(*
Nazwa:			FB_ROPPCapping
Opis:			
Wersja:			v0.1
Data:			2025-01-13
Autor:			DP
Urzadzenia:		
Konfiguracja:	
Info:
-
*)

FUNCTION_BLOCK FB_ROPPCapping
VAR_INPUT
	
	bEnable						: BOOL;					//Zezowlenie na pracę stacji sprawdzania
	bEStop						: BOOL;					//Stop Awaryjny nieaktywny
	bRun1						: BOOL;					//Włączenie 
	bRun2						: BOOL;					//Włączenie
	bRunEngine					: BOOL;					
	bHoming						: BOOL;					//Zezwolenie na wykonanie bazowania i pozycjonowania stacji sprawdzania
	bHeightSet					: BOOL;					//Bit do bazowania stacji na ustaloną wysokość 
	bIgnoreError				: BOOL;					//Ignorowania błędów cyklu pracy
	bReset						: BOOL;					//Reset błędu, jeśli w stanie "eError"
	iTime						: INT; 				
	iTime2						: INT; 				
	iTool						: INT;					//Wybór narzędzia (1-5), opisy w tablicy AsGripperScrewerTool	

	IbCapping1Tool1ActuatorUpSensor		: BOOL;		
	IbCapping1Tool1ActuatorDownSensor	: BOOL;	
	IbCapping2Tool1ActuatorUpSensor		: BOOL;	
	IbCapping2Tool1ActuatorDownSensor	: BOOL;	

	IbCapping1Tool2ActuatorUpSensor		: BOOL;		
	IbCapping1Tool2ActuatorCappingDoneSensor: BOOL;	
	IbCapping2Tool2ActuatorUpSensor			: BOOL;	
	IbCapping2Tool2ActuatorCappingDoneSensor: BOOL;	



	InEngineVelocityCV 			: UDINT;		
	InEngineSTW 				: UINT; 				// Statusword transportera wejściowo wyjściowego
	IbEngineWcState				: BOOL; 				// Statusword transportera wejściowo wyjściowego
	InEngine2VelocityCV 		: UDINT;		
	InEngine2STW 				: UINT; 				// Statusword transportera wejściowo wyjściowego
	IbEngine2WcState			: BOOL; 				// Statusword transportera wejściowo wyjściowego

	_HEIGHTMOTOR_ 				: BOOL;
	lrHeightMotorSV				: LREAL;			// Zadana wysokość
	udiHeightMotorEncoderCV		: UDINT;				// Ilość impulsów z modułu enkoderowego
	bHeightEncoderSetCDone		: BOOL;					// Zerowanie enkodera wykonane
	rHeightMotorPositionOffset 	: REAL;					// Wysokość bazowani podnośnika
	lrMaxHeight					: LREAL;				// Maksymalna wysokość podnośnika 
	lrMinHeight					: LREAL;				// Minimalna wysokość podnośnika

	bManualMovement				: BOOL; 				//Uruchomienie trybu ruchów ręcznych
	udiStationIndex				: UDINT;				// Indywidualny numer stacji
	sStationName				: STRING;				// Nazwa stacji
	
END_VAR

VAR_OUTPUT
	eState						: E_Station;			// Aktualny stan stacju
	eRunningState				: E_GripperScrewer;		// Stan pracy stacji
	eRunningStateBeforeEstop	: E_GripperScrewer;  	// Stan przed Estope
	bError						: BOOL;					// Błąd stacji
	udiErrorID					: UDINT;				// Nr blędu przeciągania formatek
	sErrorDescription			: STRING(200);			// Opis błędu
	sErrorDescription2			: STRING(200);			// Opis błędu
	sErrorStationName			: STRING;				// Nazwa stacj
	udiStationID				: UDINT;				// Nr stacji

	bHeightMotorUp				: BOOL;					//Sterowanie silnikiem podnośnika  - RUCH W GÓRĘ
	bHeightMotorDown			: BOOL;					//Sterowanie silnikiem podnośnika  - RUCH W DÓŁ
	udiHeightMotorEncoderSetCV	: UDINT;		
	bHeightEncoderSetC			: BOOL;					// Zerowanie enkodera
	lrHeightMotorCV				: LREAL;				// Aktualna pozycja podnośnika

	QnEngineVelocitySV 			: UDINT; 				// Nastawa prędkości
	QnEngineCTW 				: UINT;  				// Controlword transportera we/wy	
	QnEngine2VelocitySV 		: UDINT; 				// Nastawa prędkości
	QnEngine2CTW 				: UINT;  				// Controlword transportera we/wy	
	bHomingNeeded				: BOOL;					// Wymagane ponowne bazowanie (blad podczas bazowania lub stop awaryjny)
	bHomingDone					: BOOL;					// Stacja zbazowana 
	bCycleDone1					: BOOL;					// Sygnał o zakończeniu cyklu
	bCycleNotDone1				: BOOL;					// Sygnał o niezakończonym cyklu	
	bCycleDone2					: BOOL;					// Sygnał o zakończeniu cyklu
	bCycleNotDone2				: BOOL;					// Sygnał o niezakończonym cyklu

	tCycleTime					: TIME;	 				// Czas cyklu 
	sWarningDescription			: STRING;
	bWarning1					: BOOL;
	udiWarningID				: UDINT;
	
	bCapping1Tool1Actuator		: BOOL;
	bCapping2Tool1Actuator		: BOOL;
	bCapping12Tool1BlockActuator: BOOL;
	bCappingBlockActuator		: BOOL;
	bCapping1Tool2Down			: BOOL;		
	bCapping1Tool2Tight			: BOOL;	
	bCapping1Tool2Realese		: BOOL;	
	bCapping2Tool2Down			: BOOL;		
	bCapping2Tool2Tight			: BOOL;	
	bCapping2Tool2Realese		: BOOL;
	bFormPositioning			: BOOL;

	AsToolDescription			: ARRAY [1..10] OF STRING;	// Opis narzędzi, 1 - Opis narzędzia nr 1, 2 - Opis narzędzia nr 2
	sTool						: STRING;
	
END_VAR

VAR_IN_OUT
	
	bManualHeightMotorUp				: BOOL;					//Ruch ręczny podnośnika stacji w górę
	bManualHeightMotorDown				: BOOL;					//Ruch ręczny podnośnika stacji w dół
	bManualEngine1						: BOOL;					//Ręczne włączenie silnika sortera
	bManualEngine2						: BOOL;					//Ręczne włączenie silnika sortera
	bManualCapping1Tool1Actuator		: BOOL;
	bManualCapping2Tool1Actuator		: BOOL;
	bManualCapping12Tool1BlockActuator	: BOOL;
	bManualCappingBlockActuator			: BOOL;
	bManualCapping1Tool2Down			: BOOL;		
	bManualCapping1Tool2Tight			: BOOL;	
	bManualCapping1Tool2Realese			: BOOL;	
	bManualCapping2Tool2Down			: BOOL;		
	bManualCapping2Tool2Tight			: BOOL;	
	bManualCapping2Tool2Realese			: BOOL;
	bManualFormPositioning				: BOOL;

END_VAR

VAR
	i							:	INT;
	aBufferedSensorValue		:	ARRAY[0..50] OF BOOL;	
	iValvesCycleCase			:	INT;
	rtOutSensor					:	R_TRIG;

	// State
	eLastState					: E_Station;			//Stan ogólny bloku
	eLastStateTemp				: E_Station;			//Stan ogólny bloku
	eLastRunningState			: E_GripperScrewer;		//Stan podbloku
	eLastRunningStateTemp		: E_GripperScrewer;		//Stan podbloku

	fbHeightMotorEncoder		: FB_JiesangActuatorEncoderModul;				// Blok enkodera podnośnika chwytaka stabilizującego pod zakręcarką	
	bHeightMotorEncoderCounterReset						:BOOL; 				// Sygnał resetu enkodera
	lrLastHeightMotorPositionCV		: LREAL;				// Pozycja podnośnika w poprzednim cyklu programu
	bHeightMotorEncoderHomed	: BOOL;					// Informacja od enkodera że jest zbazowany		
	bStateError					: BOOL;
	
	tofHeightMotorDown			: TOF;					// Opóźnienie ruchu w dół, żeby nie przeciązać rozruchem układu
	rtEncoderHomed				: R_TRIG;				// Bit zakończenia enkodera
		
	tonHeightNoChange			: TON; 					// Timer wykrycia braku ruchu siłownika zmiany wysokości stacji
	tonHeightNoChangeTime		: TON; 					// Timer wykrycia braku ruchu siłownika zmiany wysokości stacji
	
	tonLimitPosMinReachedDelay	: TON;					// Timer osoiągniecia minimalnej wyskości 
	tonLimitPosMaxReachedDelay	: TON;					// Timer osiągnięcia maksymalnej wyskości
	tonSortingEngineOn			: TON;					// Opóźnienie po załączeniu napędu
	tonSortingEngineOff			: TON;					// Opóźnienie wyłączenia napędu
	tonSleeveFullEngineOn		: TON;					// Czas załączenia napędu po wykrciu braku nasadek
	tonEngineBlocked			: TON;					// Zablokowany silnik	
	rtCapSorterSensor			: R_TRIG;				// Triger
	tonTryUnblockWheel			: TON;					// Czas ruchu falownika w drugą stronę
	tofCapFeederSorterCapSensor	: TOF;					// Opóźnienie sygnału z czujnika obecności nasadki ultradzwiek
	tonCapFeederSorterCapSensor	: TON;					// Opóźnienie sygnału z czujnika obecności nasadki ultradźwięk
	tonAirBeforeStart			: TON;					// Czasówka opóźeniani przedmuchu
	tonAirBeforeStart2			: TON;					// Czasówka opóźeniani przedmuchu
	tonAirAfterStop				: TON;					// Czasówka przedmuchu po zatrzymaniu
	tonStoppingTime				: TON;					// Czasówka zbyt długiego zatrzymawania

	
	tonErrorHeightChange		: TON; 					// Timer błędu zacięcia się podnośnika
	tonMaxHeightError			: TON;					// Timer ustawienia zbyt dużej wysokości stacji
	tonMinHeightError			: TON;					// Timer ustawienia zbyt małej wysokości stacji
	tonCycleTimer				: TON;					// Czasówka cyklu
	rtrigCycleTimerRead			: R_TRIG;				// Trigger do statystyk cyklu 
	
	rtResetCommands				: R_TRIG;
	tonHomingSensor: TON;
	TimerOn: TON;
	TimerOff: TON;
	bImpOn: BOOL;
	rtCapFeederSorterCapSensor: R_TRIG;
	bBlowDelay: BOOL;
	tonbBlowDelay: TON;
	
	fbInverter: FB_MitsubishiInverter;
	fbInverter2: FB_MitsubishiInverter;	
	tonInverterError: TON;
	tonInverter2Error: TON;	
	tonbCapping1Tool2ActuatorUpError: TON;
	tonbCapping2Tool2ActuatorUpError: TON;	
	
	(*Ostrzeżenia*)
	fbbLevelSensor:	FB_InputFilter;
	(*Inne*)	

	tonGates1	:	TON;	//Czasówka dla szlabanów w rękawe
	tonGates2	:	TON;	//Czasówka dla szlabanów w rękawe
	tonGates3	:	TON;	//Czasówka dla szlabanów w rękawe
	tonGates4	:	TON;	//Czasówka dla szlabanów w rękawe

	toneHolding1 :TON;
	toneHolding2 :TON;
	toneGoingUp	:TON;
	toneHolding1Tool2 :TON;
	toneHolding2Tool2 :TON;
	
	bDone1				: BOOL;					// Sygnał o niezakończonym cyklu
	bDone2				: BOOL;					// Sygnał o niezakończonym cyklu
	
	tonDown1:TON;
	tonDown2:TON;	
	tonEnginesRun:TON;	
	tonDone	:TON;	
	ftbRunEngine: F_TRIG;
	bGates	    :	BOOL;	//Controla szłabanow w rękawe  
	bTryUnblockWheel : BOOL;
	iTryUnblockWheel : INT;
END_VAR

//Wywołanie bloczków od stacji. Ważna jest ich kolejność!!!
ACT_Limits();
ACT_HeightMotor();
ACT_ErrorHandling();

ACT_Signals();
ACT_Control();
aEngine();
ACT_Inverter();
ACT_Statistic();
ACT_Status();
ACT_Warnings();
aStationID();	

lrLastHeightMotorPositionCV:=lrHeightMotorCV;

ACTION ACT_Control:
	(*****Wyłączenie enable*****)
	IF NOT bEnable THEN
		IF eState <> E_Station.eDisabled AND eState <> E_Station.ePreparingToDisable THEN
				eState 				:= E_Station.ePreparingToDisable; 
		END_IF	
	END_IF

	(*****Estop*****)
	IF NOT bEstop  THEN	
		IF eState <> E_Station.eAborted AND eState <> E_Station.eAborting AND eState <> E_Station.eDisabled THEN
				eState 				:= E_Station.eAborting; 
		END_IF
	END_IF


	CASE eState OF
//--------------------------------------------------------------------------------
// Stan maszyny po wyłączeniu i przygotowanie do uruchomienia
	E_Station.eDisabled: 					// Stan nieaktywnosci (Stacja wyłączona) 
	
		IF bEnable THEN
			eState 				:= E_Station.ePreparingToReady; 
		END_IF 
		
//--------------------------------------------------------------------------------
// Stan maszyny po zatrzymaniu awaryjnym   
	E_Station.eAborted: 					// Stan bezpiecznego zatrzymania (po Abortingu) 

		IF bEStop THEN
			eState 				:= E_Station.ePreparingToReady;
		END_IF
		
//--------------------------------------------------------------------------------
// Stan maszyny naciśnieciu estopa 	
	E_Station.eAborting:                 	// Stan bezpiecznego zatrzymywania (po EStopie)

		ACT_ResetCommands();

		eState 						:=  E_Station.eAborted;  
		eRunningState				:=	E_GripperScrewer.eReady;
		
//--------------------------------------------------------------------------------
// Stan masyzny po wykryciu błędu			
	E_Station.eError:                 	 	// Stan błędu 	
		
		ACT_ResetCommands();
		
		IF bReset THEN
			eState 					:= E_Station.eResetting;
			bError					 := FALSE;
		END_IF
		
//--------------------------------------------------------------------------------
// Stan masyzny po wykryciu błędu
	E_Station.eResetting:					// Stan resetowania bledu (po Errorze)
			CASE udiErrorID OF
		
				//Error - Błąd falownika
				353,354:
					fbInverter.bReset	:= TRUE;
					fbInverter2.bReset	:= TRUE;					
					bError 				:= FALSE;
				ELSE
					bError := FALSE;	
			END_CASE		
		
		IF NOT bError AND fbInverter.eState = E_Station.eReady THEN
			fbInverter.bReset	:= FALSE;	
			fbInverter2.bReset	:= FALSE;
			//{warning 'Sprawdzić błąd falownika CapFeeder'}
			udiErrorID 			:=	0;
			sErrorDescription 	:=	'';
			eState 				:=	E_Station.ePreparingToReady;
			eRunningState		:=	E_GripperScrewer.eReady;
		ELSE
			eState 				:=	E_Station.eError;
		END_IF
    
//--------------------------------------------------------------------------------
// Stan ruchoow manualnych
	E_Station.eManualMovement:     			// Stan ruchów manualnych  
   
		ACT_ManualMovements();
		//Wyjście z trybu serwisowego
		IF NOT bManualMovement THEN
			bHeightMotorUp				:=	FALSE;
			bHeightMotorDown			:=	FALSE;
			eState:=E_Station.eReady;
		END_IF
		
//--------------------------------------------------------------------------------
// Stan rozpoczecia bazowania
	E_Station.eHoming:						// Stan bazowania 
		
		ACT_Homing();
		IF NOT bHoming AND NOT bHeightSet THEN
			bHeightMotorDown				:=	FALSE;
			bHeightMotorUp					:=	FALSE;
		   eState							:=	E_Station.ePreparingToReady;
		END_IF		
		
//--------------------------------------------------------------------------------
// Stan zakończenia bazowania
	E_Station.eHomingDone:                  // Stan wykonania bazowania 
	
		bHeightMotorDown					:=	FALSE;
		bHeightMotorUp						:=	FALSE;
		bHeightMotorEncoderCounterReset		:=	FALSE;
		bHomingDone							:=	TRUE;
		IF NOT bHoming AND NOT bHeightSet THEN
		   eState:=E_Station.eReady;
		END_IF
		
//--------------------------------------------------------------------------------
// Stan przygotowania do gotowości
	E_Station.ePreparingToReady:            // Stan przygotowywania do gotowosci (zawsze przed Ready)  

		eRunningState	:=	E_GripperScrewer.eReady;
		eState			:=	E_Station.eReady;	
		
//-------------------------------------------------------------------------------
// Stan przygotowania do wyłączenia maszyny
	E_Station.ePreparingToDisable:          // Stan przygotowywania do nieaktywnosci (po wyłączeniu Enable) 

		bHeightMotorUp		:=	TRUE;
		bHeightMotorDown	:=	FALSE;	
		IF tonHeightNoChange.Q OR tonHeightNoChangeTime.Q THEN
			bHeightMotorUp			:=	FALSE;
			bHeightMotorDown		:=	FALSE;	
			eRunningState			:=	E_GripperScrewer.eReady;		
			eState					:=	E_Station.eDisabled;
		END_IF	
			
//--------------------------------------------------------------------------------
// Stan gotowości
	E_Station.eReady:						// Stan gotowosci 
	
		(*Skasowanie wszystkich komend*)
		IF rtResetCommands.Q THEN	ACT_ResetCommands();	END_IF
	
		IF (bRun1 OR bRun2) AND NOT bCycleDone1 AND NOT bCycleNotDone1 AND NOT bCycleDone2 AND NOT bCycleNotDone2 THEN
			eState 				:= E_Station.eStarting; 
		END_IF
		IF bHoming OR bHeightSet THEN
			eState 				:= E_Station.eHoming; 
		END_IF
		IF bManualMovement THEN
			bManualHeightMotorUp					:=	bHeightMotorUp;					
			bManualHeightMotorDown				:=	bHeightMotorDown;	
			bManualEngine1						:=	fbInverter.bRun;							
			bManualEngine2						:=	fbInverter2.bRun;		
			bManualCapping1Tool1Actuator		:=	bCapping1Tool1Actuator;		
			bManualCapping2Tool1Actuator		:=	bCapping2Tool1Actuator;		
			bManualCapping12Tool1BlockActuator	:=	bCapping12Tool1BlockActuator;
			bManualCappingBlockActuator			:=	bCappingBlockActuator;	
			bManualCapping1Tool2Down			:=	bCapping1Tool2Down;	
			bManualCapping1Tool2Tight			:=	bCapping1Tool2Tight;			
			bManualCapping1Tool2Realese			:=	bCapping1Tool2Realese;		
			bManualCapping2Tool2Down			:=	bCapping2Tool2Down;				
			bManualCapping2Tool2Tight			:=	bCapping2Tool2Tight;
			bManualCapping2Tool2Realese			:=	bCapping2Tool2Realese;
			bManualFormPositioning				:=	bFormPositioning;			
			eState 								:=	E_Station.eManualMovement; 
		END_IF
		IF NOT bRun1 AND NOT bRun2 THEN
			bDone1						:= FALSE;
			bDone2						:= FALSE;
			bCycleDone1 				:= FALSE;
			bCycleNotDone1 				:= FALSE;	
			bCycleDone2					:= FALSE;
			bCycleNotDone2 				:= FALSE;	
			bWarning1					:= FALSE;	
		END_IF
		
//--------------------------------------------------------------------------------
// Stan zatrzymywania
	E_Station.eStopping:					// Stan zatrzymywania 
		
		ACT_Running();

		IF tonStoppingTime.Q THEN
			ACT_ResetCommands();
			eRunningState							:= E_GripperScrewer.eReady;
			eState									:= E_Station.eReady;
		END_IF

		
//--------------------------------------------------------------------------------
// Stan uruchomienia lini ( po eReady)
	E_Station.eStarting:                  	// Stan uruchamiania (po Ready)

		eState					 := E_Station.eRunning; 

//--------------------------------------------------------------------------------
// Stan wykonywania pracy
	E_Station.eRunning:               		// Stan wykonywania cyklu (po Startingu), w tym stanie osobny

		ACT_Running();
		IF NOT bRun1 AND NOT bRun2 THEN					(*Przerywanie cyklu*)
			eState 				 := E_Station.eStopping;	
		END_IF
		IF (bCycleDone1 OR bCycleNotDone1) AND (bCycleDone2 OR bCycleNotDone2)  THEN (*Cykl zakończony*)
			eState 				 := E_Station.eReady;
		END_IF						
		
		
END_CASE
END_ACTION

ACTION ACT_ErrorHandling:
//OBSŁUGA BŁĘDÓW STACJI SPRAWDZANIA
//************LISTA BŁĘDÓW***************
bStateError:= (eState=E_Station.eError) OR (eState=E_Station.eResetting) OR bIgnoreError;
//************LISTA BŁĘDÓW***************

//Error 1 - podnośnik nie porusza się pomimo wysterowania 
tonErrorHeightChange(IN:=(bHeightMotorUp OR bHeightMotorDown) AND lrLastHeightMotorPositionCV=lrHeightMotorCV, PT:=T#3S);
tonMaxHeightError	(IN:=lrHeightMotorSV>lrMaxHeight AND NOT bHomingNeeded AND eState=E_Station.eReady,PT:=T#30S);
tonMinHeightError	(IN:=lrHeightMotorSV<lrMinHeight AND NOT bHomingNeeded AND eState=E_Station.eReady,PT:=T#30S);
tonInverterError	(IN:=fbInverter.bError AND NOT bStateError, PT:=T#3S);
tonInverter2Error	(IN:=fbInverter2.bError AND NOT bStateError, PT:=T#3S);

tonbCapping1Tool2ActuatorUpError (IN:= iTool = 2 (*G.dociskająca*) AND NOT IbCapping1Tool2ActuatorUpSensor AND NOT bCapping1Tool2Down, PT:=T#2S);
tonbCapping2Tool2ActuatorUpError (IN:= iTool = 2 (*G.dociskająca*) AND NOT IbCapping2Tool2ActuatorUpSensor AND NOT bCapping2Tool2Down, PT:=T#2S);

IF (bEnable OR (eState = E_Station.ePreparingToDisable)) AND NOT bIgnoreError THEN
	
	IF tonErrorHeightChange.Q THEN
		bError:=TRUE;
		udiErrorID:=350;
		sErrorDescription:='Blokada podnośnika lub brak zasilania - sprawdź czujnik lub odblokuj mechanicznie';	
		sErrorDescription2:='';
	END_IF
	
	//Error - Bład nastaw max
	IF tonMaxHeightError.Q  THEN
		bError:=TRUE;
		udiErrorID:=351;
		sErrorDescription:='Wartość zadana wysokości jest większa od maksymalnej - zmień ustawienia w recepturze';
		sErrorDescription2:=REAL_TO_STRING(LREAL_TO_INT(lrMaxHeight));
	END_IF
	
	//Error - Bład nastaw min
	IF tonMinHeightError.Q THEN
		bError:=TRUE;
		udiErrorID:=352;
		sErrorDescription:='Wartość zadana wysokości jest mniejsza od minimalnej - zmień ustawienia w recepturze';
		sErrorDescription2:=REAL_TO_STRING(LREAL_TO_INT(lrMinHeight));
	END_IF	
	
	//Error - Bład falownika 1
	IF tonInverterError.Q THEN
		bError:=TRUE;
		udiErrorID:=353;
		sErrorDescription:='Błąd falownika głowicy 1';
		sErrorDescription2:='';
	END_IF		
	
	//Error - Bład falownika 2
	IF tonInverter2Error.Q THEN
		bError:=TRUE;
		udiErrorID:=354;
		sErrorDescription:='Błąd falownika głowicy 2';
		sErrorDescription2:='';
	END_IF			
	
	//Error Glowica 1 - Bład góry
	IF tonbCapping1Tool2ActuatorUpError.Q THEN
		bError:=TRUE;
		udiErrorID:=355;
		sErrorDescription:='Błąd górnej pozycji głowicy dociskającej 1- upewnij się że jest wybrane dobre narzędzie lub sprawdź czujnik';
		sErrorDescription2:='';	
	END_IF			
	//Error Glowica 2 - Bład góry
	IF tonbCapping2Tool2ActuatorUpError.Q THEN
		bError:=TRUE;
		udiErrorID:=356;
		sErrorDescription:='Błąd górnej pozycji głowicy dociskającej 2 - upewnij się że jest wybrane dobre narzędzie lub sprawdź czujnik';
		sErrorDescription2:='';	
	END_IF			
	
ELSE
	bError	:=FALSE;
END_IF


//-----------------------------------------------------------------------
IF bError AND NOT bStateError THEN

	IF eLastState = eRunning THEN
		bCycleNotDone1						:= TRUE;
	END_IF

	eState 									:= E_Station.eError;
END_IF


//------------------------------------------------------------------------

(*Wyświetlanie błedu na wyjściu*)
bError;

(*Przepisywanie nazwy stacji*)
sErrorStationName 							:= sStationName;

//Jezeli nie zbazowane to potrzebne bazowanie
IF NOT bHeightMotorEncoderHomed  THEN
	bHomingDone								:=	FALSE;
END_IF
END_ACTION

ACTION ACT_HeightMotor:
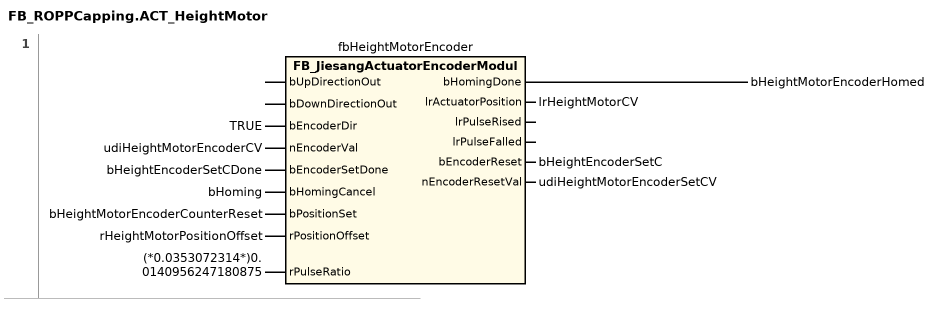
// NETWORK 1
fbHeightMotorEncoder(
    bEncoderDir := TRUE,
    nEncoderVal := udiHeightMotorEncoderCV,
    bEncoderSetDone := bHeightEncoderSetCDone,
    bHomingCancel := bHoming,
    bPositionSet := bHeightMotorEncoderCounterReset,
    rPositionOffset := rHeightMotorPositionOffset,
    rPulseRatio := (*0.0353072314*)0.0140956247180875,
    lrActuatorPosition => lrHeightMotorCV,
    bEncoderReset => bHeightEncoderSetC,
    nEncoderResetVal => udiHeightMotorEncoderSetCV); // FB_JiesangActuatorEncoderModul
bHeightMotorEncoderHomed := fbHeightMotorEncoder.bHomingDone;
END_ACTION

ACTION ACT_Homing:
//BAZOWANIE

tofHeightMotorDown(IN:=bHeightMotorDown, PT:=T#1S); //Zabezpieczenie przed zbyt szybkim przełączeniem pomiędzy Down a Up, bezpiecznieki sie palą
	
//Podnoszenie stacji do maksymalnej pozycji
IF NOT bHeightMotorEncoderHomed OR rtEncoderHomed.Q THEN
	bHeightMotorUp:=(*TRUE*) NOT tofHeightMotorDown.Q AND NOT tonHomingSensor.Q;
	bHeightMotorDown:=FALSE;
	IF tonHeightNoChange.Q OR tonHeightNoChangeTime.Q THEN
		bHeightMotorEncoderCounterReset:=TRUE;
		bHeightMotorUp:=FALSE;
    END_IF
	//Jesli enkoder zbazowany zakończ bazowanie	
	IF rtEncoderHomed.Q  THEN
		bHeightMotorUp:=FALSE;
		bHeightMotorDown:=FALSE;
		eState:=E_Station.eHomingDone;
	END_IF		
		
//Po podniesieniu stacji opuszczanie do ustalonej wysokości
ELSIF bHeightMotorEncoderHomed THEN
	bHeightMotorEncoderCounterReset:=FALSE;
	bHeightMotorUp:=lrHeightMotorCV<=lrHeightMotorSV;
	bHeightMotorDown:=lrHeightMotorCV>=lrHeightMotorSV;
	//Kiedy stacja osiągnie wysokość zadaną
	IF ABS(lrHeightMotorCV-lrHeightMotorSV)<0.5 OR tonLimitPosMaxReachedDelay.Q OR tonLimitPosMinReachedDelay.Q THEN
		bHeightMotorDown:=FALSE;
		bHeightMotorUp:=FALSE;
		eState:=E_Station.eHomingDone;
	END_IF			
END_IF
END_ACTION

ACTION ACT_Inverter:
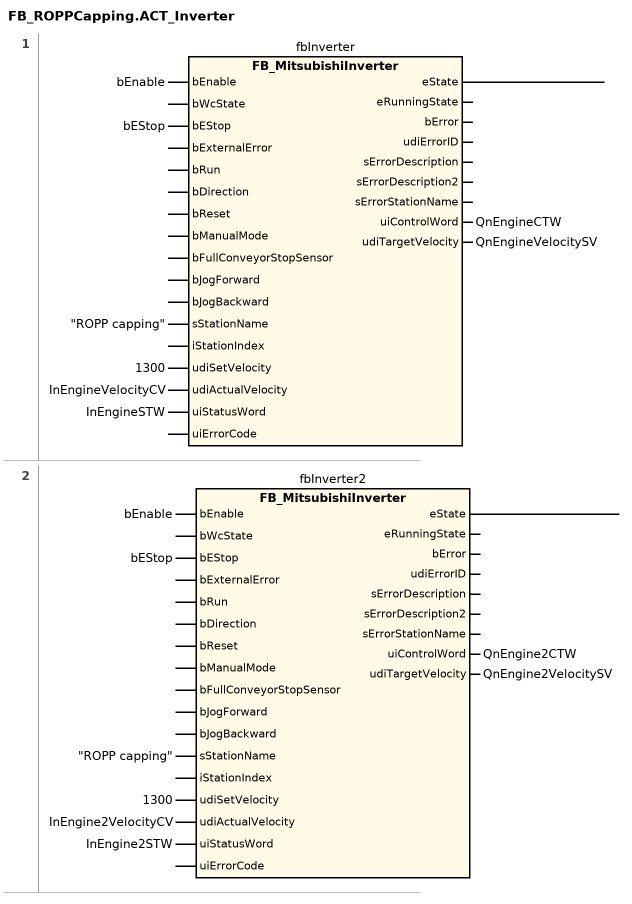
// NETWORK 1
fbInverter(
    bEnable := bEnable,
    bEStop := bEStop,
    sStationName := "ROPP capping",
    udiSetVelocity := 1300,
    udiActualVelocity := InEngineVelocityCV,
    uiStatusWord := InEngineSTW,
    uiControlWord => QnEngineCTW,
    udiTargetVelocity => QnEngineVelocitySV); // FB_MitsubishiInverter

// NETWORK 2
fbInverter2(
    bEnable := bEnable,
    bEStop := bEStop,
    sStationName := "ROPP capping",
    udiSetVelocity := 1300,
    udiActualVelocity := InEngine2VelocityCV,
    uiStatusWord := InEngine2STW,
    uiControlWord => QnEngine2CTW,
    udiTargetVelocity => QnEngine2VelocitySV); // FB_MitsubishiInverter
END_ACTION

ACTION ACT_Limits:

END_ACTION

ACTION ACT_ManualMovements:
//W trybie ruchów manualnych wykonuj ruchy za pomocą rozkazów manualnych
IF NOT bRun1 AND NOT bRun2 THEN
	
	bHeightMotorUp					:=	bManualHeightMotorUp;				
	bHeightMotorDown				:=	bManualHeightMotorDown;				
	fbInverter.bRun					:=	bManualEngine1;						
	fbInverter2.bRun				:=	bManualEngine2;						
	bCapping1Tool1Actuator			:=	bManualCapping1Tool1Actuator;		
	bCapping2Tool1Actuator			:=	bManualCapping2Tool1Actuator;		
	bCapping12Tool1BlockActuator	:=	bManualCapping12Tool1BlockActuator OR bManualCapping1Tool1Actuator OR bManualCapping2Tool1Actuator;	
	bCappingBlockActuator			:=	bManualCappingBlockActuator ;//OR bManualCapping1Tool1Actuator OR bManualCapping2Tool1Actuator;			
	bCapping1Tool2Down				:=	bManualCapping1Tool2Down;			
	bCapping1Tool2Tight				:=	bManualCapping1Tool2Tight;			
	bCapping1Tool2Realese			:=	bManualCapping1Tool2Realese;			
	bCapping2Tool2Down				:=	bManualCapping2Tool2Down;			
	bCapping2Tool2Tight				:=	bManualCapping2Tool2Tight;			
	bCapping2Tool2Realese			:=	bManualCapping2Tool2Realese;			
	bFormPositioning				:=	bManualFormPositioning;				

ELSE	//Kasuje zeby po cyklu nic sie nie poruszało

	bManualHeightMotorUp				:= FALSE;		
	bManualHeightMotorDown				:= FALSE;		
	bManualEngine1						:= FALSE;	
	bManualEngine2						:= FALSE;	
	bManualCapping1Tool1Actuator		:= FALSE;	
	bManualCapping2Tool1Actuator		:= FALSE;	
	bManualCapping12Tool1BlockActuator	:= FALSE;	
	bManualCappingBlockActuator			:= FALSE;	
	bManualCapping1Tool2Down			:= FALSE;	
	bManualCapping1Tool2Tight			:= FALSE;	
	bManualCapping1Tool2Realese			:= FALSE;	
	bManualCapping2Tool2Down			:= FALSE;	
	bManualCapping2Tool2Tight			:= FALSE;	
	bManualCapping2Tool2Realese			:= FALSE;	
	bManualFormPositioning				:= FALSE;	

END_IF

IF bHoming OR bHeightSet THEN
	eState:=E_Station.eHoming;
END_IF

IF bRun1 OR bRun2 THEN	
	ACT_Running();
END_IF

IF NOT bRun1 AND NOT bRun2 THEN
	bCycleDone1 				:= FALSE;
	bCycleNotDone1 				:= FALSE;	
	bCycleDone2					:= FALSE;
	bCycleNotDone2 				:= FALSE;	
	bWarning1					:= FALSE;	
END_IF

//Zabezpieczenie przed kolizją stacji poprzez ruch podnośnika	
IF bHeightMotorDown AND lrHeightMotorCV<=lrMinHeight AND NOT bHoming AND NOT bHeightSet THEN
	bHeightMotorDown:=FALSE;
END_IF	

IF bHeightMotorUp AND lrHeightMotorCV>=lrMaxHeight AND NOT bHoming AND NOT bHeightSet THEN
	bHeightMotorUp:=FALSE;
END_IF
END_ACTION

ACTION ACT_ResetCommands:
//Reset komend ruchu 	

bHeightMotorUp					:=	FALSE;
bHeightMotorDown				:=	FALSE;
fbInverter.bRun					:=	FALSE;
fbInverter2.bRun				:=	FALSE;
bCapping1Tool1Actuator			:=	FALSE;
bCapping2Tool1Actuator			:=	FALSE;
bCapping12Tool1BlockActuator	:=	FALSE;
bCappingBlockActuator			:=	FALSE;
bCapping1Tool2Down				:=	FALSE;
bCapping1Tool2Tight				:=	FALSE;
bCapping1Tool2Realese			:=	FALSE;
bCapping2Tool2Down				:=	FALSE;
bCapping2Tool2Tight				:=	FALSE;
bCapping2Tool2Realese			:=	FALSE;
bFormPositioning				:=	FALSE;
END_ACTION

ACTION ACT_Running:

CASE eRunningState OF

//====================================
	
	(*Oczekiwanie na wykonanie pojedynczego cyklu*)
	E_GripperScrewer.eReady:
	 		                                       	
		IF NOT bCycleDone1 AND NOT bCycleNotDone1 AND NOT bCycleDone2 AND NOT bCycleNotDone2 THEN                                           	
			IF bRun1 OR bRun2 THEN                			
					eRunningState						:=	E_GripperScrewer.eToPushingPosition;	
			END_IF
		END_IF
		
//====================================		
	(*Ruch na pozycję *)			
	E_GripperScrewer.eToPushingPosition:
	
		bFormPositioning				:= TRUE;
	
		bCapping12Tool1BlockActuator	:= TRUE;
		bCappingBlockActuator			:= TRUE;	
		
		IF		iTOOL = 1 THEN //Glowica zakręcająca
			fbInverter.bRun				:= bRun1;
			fbInverter2.bRun			:= bRun2;	

			IF bManualMode AND tonEnginesRun.Q THEN
				bCapping1Tool1Actuator		:= bRun1;
				bCapping2Tool1Actuator		:= bRun2;	
				eRunningState				:=	E_GripperScrewer.eScrewing;	
			ELSIF NOT bManualMode THEN
				bCapping1Tool1Actuator		:= bRun1;
				bCapping2Tool1Actuator		:= bRun2;	
				eRunningState				:=	E_GripperScrewer.eScrewing;	
			END_IF
			
		ELSIF	iTOOL = 2 THEN //Glowica dociskająca
			bCapping1Tool2Down			:= bRun1;	
			bCapping1Tool2Tight			:= FALSE;
			bCapping2Tool2Down			:= bRun2;
			bCapping2Tool2Tight			:= FALSE;
			eRunningState				:=	E_GripperScrewer.eScrewing;	
		END_IF
	

//====================================		
		
	(*Zakręcanie*)
	E_GripperScrewer.eScrewing:
	
		IF		iTOOL = 1 THEN //Glowica zakręcająca
			eRunningState					:=	E_GripperScrewer.eHolding;	
			
		ELSIF	iTOOL = 2 THEN //Glowica dociskająca
			
			IF tonDown1.Q THEN
				bCapping1Tool2Down			:=	bRun1;	
				bCapping1Tool2Tight			:=	bRun1;
				bCapping2Tool2Down			:=	bRun2;
				bCapping2Tool2Tight			:=	bRun2;
				eRunningState				:=	E_GripperScrewer.eHolding;
			END_IF
			
		END_IF	
	
//====================================

	(*Przytrzymanie / Czas na odbpuszczenie chwytakow*)					
	E_GripperScrewer.eHolding:
	
	
		IF		iTOOL = 1 THEN //Glowica zakręcająca
			IF (toneHolding1.Q OR NOT bRun1) THEN
				bDone1					:=	TRUE;
				bCapping1Tool1Actuator	:=	FALSE;
			END_IF
			IF (toneHolding2.Q OR NOT bRun2) THEN
				bDone2					:=	TRUE;				
				bCapping2Tool1Actuator	:=	FALSE;	
			END_IF	
			IF NOT 	bCapping1Tool1Actuator	AND NOT bCapping2Tool1Actuator THEN
				eRunningState					:=	E_GripperScrewer.eGoingUp;	
			END_IF
		ELSIF	iTOOL = 2 THEN //Glowica dociskająca

			IF (toneHolding1Tool2.Q OR IbCapping1Tool2ActuatorCappingDoneSensor OR NOT bRun1) THEN	
				bDone1						:=	IbCapping1Tool2ActuatorCappingDoneSensor;
				bCapping1Tool2Tight			:=	FALSE;
			END_IF
			
			IF (toneHolding2Tool2.Q OR IbCapping2Tool2ActuatorCappingDoneSensor OR NOT bRun2) THEN
				bDone2						:=	IbCapping2Tool2ActuatorCappingDoneSensor;		
				bCapping2Tool2Tight			:=	FALSE;
			END_IF	
			
			IF NOT 	bCapping1Tool2Tight	AND NOT bCapping2Tool2Tight THEN
				eRunningState				:=	E_GripperScrewer.eGoingUp;	
			END_IF			
	
		END_IF	

//====================================	

	(*Podnoszenie do góry / reset laga i obrót do pozycji gotowości*)			 
	E_GripperScrewer.eGoingUp:
	

		IF		iTOOL = 1 THEN //Glowica zakręcająca
			

			bCapping1Tool1Actuator			:=	FALSE;
			bCapping2Tool1Actuator			:=	FALSE;	
			bFormPositioning				:=	FALSE;			

			IF bManualMode THEN
				IF tonDone.Q THEN
					bCapping12Tool1BlockActuator	:= FALSE;
					bCappingBlockActuator			:= FALSE;
					fbInverter.bRun					:= FALSE;
					fbInverter2.bRun				:= FALSE;	
					eRunningState 					:=	E_GripperScrewer.eDone;					
				END_IF	
			ELSIF NOT bManualMode THEN	
					IF NOT bRunEngine THEN
						fbInverter.bRun					:= FALSE;
						fbInverter2.bRun				:= FALSE;	
						bCappingBlockActuator			:= FALSE;					
						eRunningState 					:=	E_GripperScrewer.eDone;	
					ELSE
						eRunningState 					:=	E_GripperScrewer.eDone;	
					END_IF			
			END_IF
		
		
		ELSIF	iTOOL = 2 THEN //Glowica dociskająca
			bCapping1Tool2Tight			:=	FALSE;		
			bCapping2Tool2Tight			:=	FALSE;	
	
			IF toneGoingUp.Q THEN
				bCapping1Tool2Down			:=	FALSE;		
				bCapping2Tool2Down			:=	FALSE;	
				eRunningState				:=	E_GripperScrewer.eDone;	
			END_IF
	
		END_IF	
		

		
//====================================			
	(*Zakręcono*)			
	E_GripperScrewer.eDone:
	
		bCycleDone1 						:=	bRun1 AND bDone1;
		bCycleNotDone1						:=	NOT bRun1 OR NOT bDone1;
		bCycleDone2 						:=	bRun2 AND bDone2;
		bCycleNotDone2						:=	NOT bRun2 OR NOT bDone2;	
	
		eRunningState 					:=	E_GripperScrewer.eReady;					


//====================================	
			
	E_GripperScrewer.eNotDone:

		bCycleNotDone1 						:=	TRUE;
		bCycleNotDone2						:=	TRUE;
		eRunningState						:=	E_GripperScrewer.eReady;	
	
END_CASE
END_ACTION

ACTION ACT_Signals:
(** Timery na potrzeby bazowania**)
rtEncoderHomed(CLK:=bHeightMotorEncoderHomed,Q=>);
tonHeightNoChange(IN:=((bHeightMotorUp OR bHeightMotorDown OR tonHomingSensor.Q) AND (lrLastHeightMotorPositionCV=lrHeightMotorCV)), PT:=T#500MS); 


tonLimitPosMinReachedDelay(IN:=(lrHeightMotorCV<=lrMinHeight) AND eState=E_Station.eHoming,PT:=T#2S);
tonLimitPosMaxReachedDelay(IN:=(lrHeightMotorCV>=lrMaxHeight) AND eState=E_Station.eHoming,PT:=T#2S);

rtResetCommands			(CLK:=	eState = E_Station.eReady (* OR *)		,Q=>); //Triger do resetu zmienych


(** Timery używane podczas pracy stacji**)
toneHolding1	(IN:=	eRunningState=E_GripperScrewer.eHolding AND IbCapping1Tool1ActuatorDownSensor, PT:= INT_TO_TIME(iTime));
toneHolding2	(IN:=	eRunningState=E_GripperScrewer.eHolding AND IbCapping2Tool1ActuatorDownSensor, PT:= INT_TO_TIME(iTime));	

toneHolding1Tool2	(IN:=	eRunningState=E_GripperScrewer.eHolding AND bCapping1Tool2Down, PT:= INT_TO_TIME(2000));
toneHolding2Tool2	(IN:=	eRunningState=E_GripperScrewer.eHolding AND bCapping2Tool2Down, PT:= INT_TO_TIME(2000));	

toneGoingUp			(IN:=	eRunningState=E_GripperScrewer.eGoingUp , PT:= T#300MS);	


tonDown1		(IN:=	eRunningState=E_GripperScrewer.eScrewing, PT:= INT_TO_TIME(iTime2));
tonDown2		(IN:=	eRunningState=E_GripperScrewer.eScrewing, PT:= INT_TO_TIME(iTime2));	

tonEnginesRun	(IN:= fbInverter.bRun OR fbInverter2.bRun, PT:=T#1S);
tonDone			(IN:= eRunningState = E_GripperScrewer.eGoingUp, PT:=T#1S);

ftbRunEngine	(CLK:=bRunEngine,Q=>);

(** Dodatkowy timer przy zatrzymywaniu**)
tonStoppingTime( IN:= eState= E_Station.eStopping, PT:=T#2S);
END_ACTION

ACTION ACT_Statistic:
//Statystyka do zliczania czasu cyklu 
rtrigCycleTimerRead(CLK:=eRunningState=E_GripperScrewer.eDone );

	IF rtrigCycleTimerRead.Q THEN
		tCycleTime:=tonCycleTimer.ET;
		
	END_IF
	
	tonCycleTimer(IN:=eRunningState>E_GripperScrewer.eReady,PT:=T#1D);
END_ACTION

ACTION ACT_Status:

(*Zapisywanie ostatniego stanu*)
	IF eLastStateTemp<>eState THEN
		eLastState := eLastStateTemp;
	END_IF
	eLastStateTemp := eState;
	
	IF eLastRunningStateTemp<>eRunningState THEN
		eLastRunningState := eLastRunningStateTemp;
	END_IF
	eLastRunningStateTemp := eRunningState;
(*Koniec Zapisywanie ostatniego stanu*)
END_ACTION

ACTION ACT_Warnings:

END_ACTION

ACTION aEngine:

IF bRunEngine THEN
	fbInverter.bRun				:=	TRUE;	
	fbInverter2.bRun			:=	TRUE;		
	bCappingBlockActuator		:=	TRUE;
END_IF

IF ftbRunEngine.Q THEN
	fbInverter.bRun				:=	FALSE;	
	fbInverter2.bRun			:=	FALSE;		
	bCappingBlockActuator		:=	FALSE;
END_IF
END_ACTION

ACTION aStationID:
udiStationID	:=	udiStationIndex;
END_ACTION

END_FUNCTION_BLOCK

(* stored: Version 1.1.0.1, ProductVersion 3.1.4026.13, FileIdentifier 94e10d7b8e8d3cbbb9327c81c4bb1d20f3551d21, FileSignature 0f960e986c8510f9d3bf5aab1cca4462ae971f155e212c335b806ebcc3f05877b503575d0bbb150d99886e23b244cc8b02d39f8c39927337cf10352bea92ee536f82a3ad4a89aef00c7877df8f5995d34a0ccd31986a9566139c569e36e5eb648b25a505c3d331d43e19e40a003664b0bd684248800c7c3abec03324e8efe928be3e2fce9385ba6bb886a72a909ce1f59c55e817cea5256ce0149f88fe3e37324fa473d7ac4f7b3ec1e99ac409c5ee8ee37de61ac1011b277410704abb0d1cda84b81713d580bc7ddf957aceac6d5460223f880d0f86db9799c489449739ab63e0e9c20ceeebd96d7a35c0b79e7d9b5b6c4f598a435e4b9eb6ab31dfa2ebead6
   POU FB_ROPPCapping: Id {5f3ec85e-4b52-4e92-a2ba-285d47a71459}, SpecialFunc None
   Action ACT_Control: Id {91fa008f-6a2e-45fe-a67d-695c1ae2a0af}
   Action ACT_ErrorHandling: Id {9a947482-57ca-4b05-983c-92ff1d2c4d87}
   Action ACT_HeightMotor: Id {ca6dc0e0-26c6-4f3d-bbed-be35749f55d2}
   Action ACT_Homing: Id {2a5fa702-17d3-4fe4-95e6-8b83ff08a018}
   Action ACT_Inverter: Id {f49d5ee5-2f3d-40f8-9093-2d6661687f26}
   Action ACT_Limits: Id {7e09d7a8-7670-4732-a2fe-0783d53254fd}
   Action ACT_ManualMovements: Id {11634e39-d51b-41d3-9708-005f4a218052}
   Action ACT_ResetCommands: Id {8739b41a-a105-43a8-9e3d-b7b034694e25}
   Action ACT_Running: Id {1ea73fb6-6de3-4695-b504-f9fee60eaa4a}
   Action ACT_Signals: Id {fcf8ba3e-0193-4a5b-ab7a-7da93bffc936}
   Action ACT_Statistic: Id {6ac5f478-f59e-4d5c-80ca-0fe051a946cc}
   Action ACT_Status: Id {9c58677c-843b-44db-898c-73fcb413d764}
   Action ACT_Warnings: Id {54c3789f-5437-44fb-b91c-60bf0ac026a2}
   Action aEngine: Id {f0d9ea7d-9156-409a-a274-f72874eb8d2a}
   Action aStationID: Id {8b42676b-6ca9-4977-bad7-628366eb354e} *)
